// TIA Portal V16 export
// export: Created 2021-07-12T14:47:14.8665105Z, ExportSetting WithDefaults, DisplayName Totally Integrated Automation Portal, DisplayVersion V16, DisplayName TIA Portal Version Control Interface, DisplayVersion V16, DisplayName TIA Portal Openness, DisplayVersion V16, DisplayName STEP 7 Professional, DisplayVersion V16, DisplayName STEP 7 Safety, DisplayVersion V16, DisplayName WinCC Professional, DisplayVersion V16
DATA_BLOCK "MasterCharacteristics_01"   // DB6001
{ S7_Optimized_Access := 'TRUE' }
FAMILY : SimaHydTO
VERSION : 1.0
// stored: AutoNumber true, DBAccessibleFromOPCUA true, InstanceOfName LSimaHydTO_typeVCharData, InstanceOfType UDT, IsOnlyStoredInLoadMemory false, IsWriteProtectedInAS false
"LSimaHydTO_typeVCharData"
   // VAR
   //    QOutput { S7_SetPoint := 'True'} : Array[0.."LSIMAHYD_VCHAR_POINTS_UPPER_LIMIT"] of Real;
   //    Velocity { S7_SetPoint := 'True'} : Array[0.."LSIMAHYD_VCHAR_POINTS_UPPER_LIMIT"] of Real;
   //    VelocityLimitPositive { S7_SetPoint := 'True'} : Real := 100.0;
   //    VelocityLimitNegative { S7_SetPoint := 'True'} : Real := -100.0;
   //    ZeroZonePositive { S7_SetPoint := 'True'} : Real;
   //    ZeroZoneNegative { S7_SetPoint := 'True'} : Real;
   //    MaxIdx { S7_SetPoint := 'True'} : Int := 4;
   //    "Name" { S7_SetPoint := 'True'} : WString[24] := 'MasterCharacteristics_01';
   // END_VAR
BEGIN
   QOutput[0] := -100.0;
   QOutput[1] := -50.0;
   QOutput[2] := 0.0;
   QOutput[3] := 50.0;
   QOutput[4] := 100.0;
   Velocity[0] := -100.0;
   Velocity[1] := -30.0;
   Velocity[2] := 0.0;
   Velocity[3] := 40.0;
   Velocity[4] := 100.0;
END_DATA_BLOCK
